// TIA Portal V19 export
TYPE "OOAx_Wng"
// stored: Access Published
   STRUCT
      SwLimitMinus : Bool;
      SwLimitPlus : Bool;
   END_STRUCT;
END_TYPE
